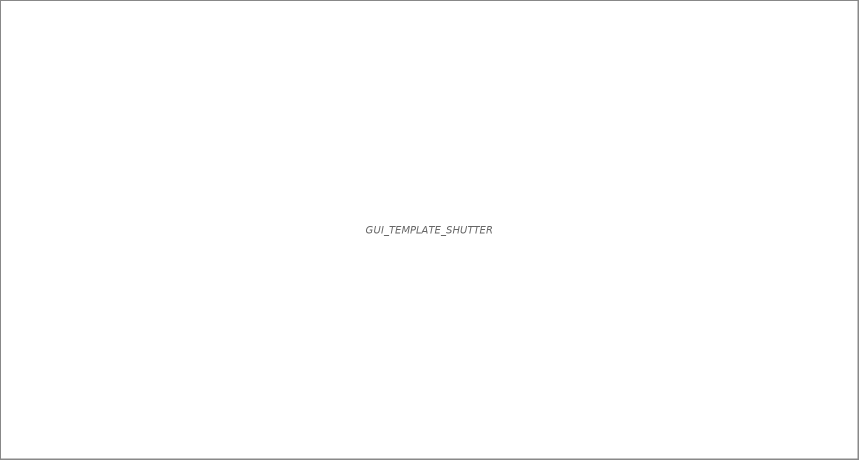
VISUALIZATION GUI_Shutter001  // 859x460
    Frame (0,0 859x460)
        shows GUI_TEMPLATE_SHUTTER(m_Instance := MAIN.Shutter001)
END_VISUALIZATION

(* stored: Version 1.1.0.1, ProductVersion 3.1.4024.3
   Visu GUI_Shutter001: Id {05fa3a21-cc3f-46e4-a133-64595b3fadfd} *)
